PROGRAM MAIN
VAR
	cntr	: INT;
	
END_VAR

cntr := cntr + 100;

END_PROGRAM

(* stored: Version 1.1.0.1
   POU MAIN: Id {2631033a-e591-4419-946a-73843d4781c2}, SpecialFunc None *)
